(* Logix 5000 project; controller Emulate Emulate 5570 rev 30.12; software revision 30.00 *)

TASK MainTask (continuous, watchdog 500 ms) : MainProgram

MODULES
   Local : Emulate 5570 (ICP 2, rev 30.12)
      VIRTUAL_INPUTS : vendor 1 type 0 code 15 (ICP 3, rev 1.1, Output RPI 50 ms)
      VIRTUAL_OUTPUTS : vendor 1 type 0 code 15 (ICP 4, rev 1.1, Output RPI 50 ms)
END_MODULES

VAR_GLOBAL   (* controller tags *)
   C_S4 : COUNTER;
   C_S5 : COUNTER;
   C_S6 : COUNTER;
   FIO_A2 : BOOL;
   FIO_B1 : BOOL;
   FIO_B2 : BOOL;
   FIO_B3 : BOOL;
   FIO_B4 : BOOL;
   FIO_Banda1 : BOOL;
   FIO_C1 : BOOL;
   FIO_RESET : BOOL;
   FIO_S1 : BOOL;
   FIO_S2 : BOOL := 1;
   FIO_S3 : BOOL;
   FIO_S4 : BOOL;
   FIO_S5 : BOOL;
   FIO_S6 : BOOL := 1;
   FIO_SB1 : BOOL;
   MOTOR : ALIAS FOR Local:4:O.Data[0].0;
   MOTOR_START : ALIAS FOR Local:3:I.Data[1].0;
   MOTOR_STOP : ALIAS FOR Local:3:I.Data[1].1;
END_VAR

PROGRAM MainProgram   (* main routine MainRoutine *)
VAR
   FIO_HMI_START : BOOL := 1;
   FIO_HMI_STOP : BOOL; {access Read Only}
   Valvula : BOOL;
END_VAR

ROUTINE MainRoutine   (* ladder *)
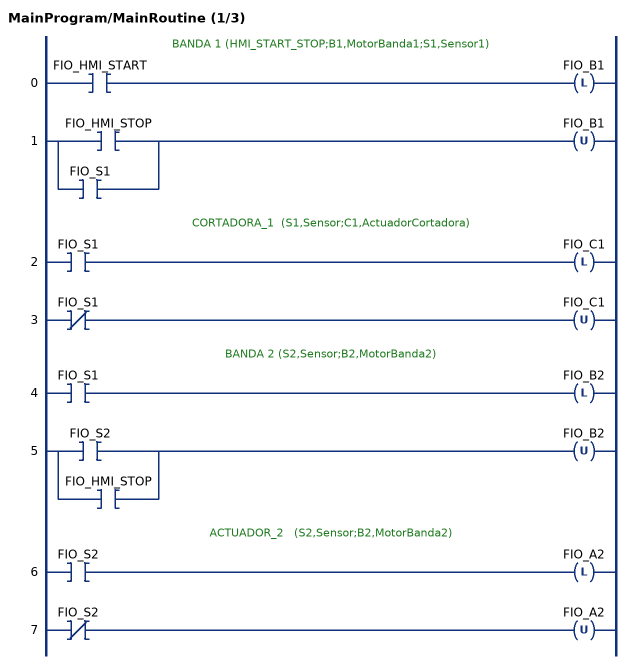
   // BANDA 1 (HMI_START_STOP;B1,MotorBanda1;S1,Sensor1)
   0: XIC(FIO_HMI_START)OTL(FIO_B1);
   1: [XIC(FIO_HMI_STOP) ,XIC(FIO_S1) ]OTU(FIO_B1);
   // CORTADORA_1  (S1,Sensor;C1,ActuadorCortadora)
   2: XIC(FIO_S1)OTL(FIO_C1);
   3: XIO(FIO_S1)OTU(FIO_C1);
   // BANDA 2 (S2,Sensor;B2,MotorBanda2)
   4: XIC(FIO_S1)OTL(FIO_B2);
   5: [XIC(FIO_S2) ,XIC(FIO_HMI_STOP) ]OTU(FIO_B2);
   // ACTUADOR_2   (S2,Sensor;B2,MotorBanda2)
   6: XIC(FIO_S2)OTL(FIO_A2);
   7: XIO(FIO_S2)OTU(FIO_A2);
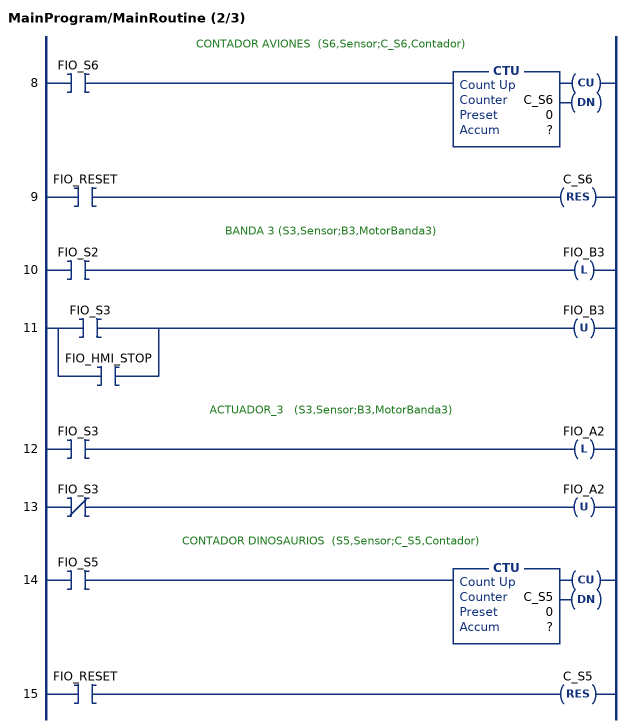
   // CONTADOR AVIONES  (S6,Sensor;C_S6,Contador)
   8: XIC(FIO_S6)CTU(C_S6,?,?);
   9: XIC(FIO_RESET)RES(C_S6);
   // BANDA 3 (S3,Sensor;B3,MotorBanda3)
   10: XIC(FIO_S2)OTL(FIO_B3);
   11: [XIC(FIO_S3) ,XIC(FIO_HMI_STOP) ]OTU(FIO_B3);
   // ACTUADOR_3   (S3,Sensor;B3,MotorBanda3)
   12: XIC(FIO_S3)OTL(FIO_A2);
   13: XIO(FIO_S3)OTU(FIO_A2);
   // CONTADOR DINOSAURIOS  (S5,Sensor;C_S5,Contador)
   14: XIC(FIO_S5)CTU(C_S5,?,?);
   15: XIC(FIO_RESET)RES(C_S5);
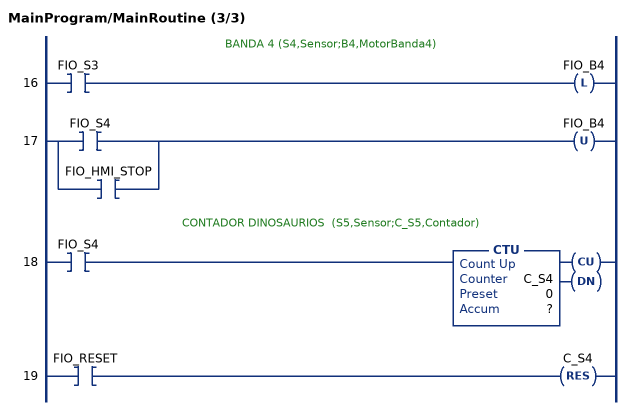
   // BANDA 4 (S4,Sensor;B4,MotorBanda4)
   16: XIC(FIO_S3)OTL(FIO_B4);
   17: [XIC(FIO_S4) ,XIC(FIO_HMI_STOP) ]OTU(FIO_B4);
   // CONTADOR DINOSAURIOS  (S5,Sensor;C_S5,Contador)
   18: XIC(FIO_S4)CTU(C_S4,?,?);
   19: XIC(FIO_RESET)RES(C_S4);
END_ROUTINE
END_PROGRAM
